// TIA Portal V18 export
FUNCTION_BLOCK "00_Push-Button_Input"   // FB9, F_LAD
{ S7_Optimized_Access := 'TRUE' }
   VAR_INPUT
      Bypass_ET200 : Bool;
      IN_1 : Bool;
      IN_2 : Bool;
      IN_3 : Bool;
      IN_4 : Bool;
      ON_Tristate : Bool;
      NormOpenDiag : Bool;   // if 1-> diag has NO logic, if 0 diag has NC logic
      ON_Lamp : Bool;
      RESET : Bool;
      REAC_DELAY { ExternalWritable := 'False'} : Time;   // Reactivation delay= the OUT goes from 0 to 1 after this time
      BLINK_CYCLE_TIME : Time := t#1250ms;
      ON_TIME : Time := T#625ms;
   END_VAR
   VAR_OUTPUT
      OUT_1 : Bool;
      OUT_2 : Bool;
      OUT_3 : Bool;
      OUT_4 : Bool;
      Diag_1 : Bool;
      Diag_2 : Bool;
      Diag_3 : Bool;
      Diag_4 : Bool;
      Lamp_1 : Bool;
      Lamp_2 : Bool;
      Lamp_3 : Bool;
      Lamp_4 : Bool;
   END_VAR
   VAR
      TON_1 { ExternalWritable := 'False'} : TON;
      TON_2 { ExternalWritable := 'False'} : TON;
      TON_3 { ExternalWritable := 'False'} : TON;
      TON_4 { ExternalWritable := 'False'} : TON;
      TOF_Lamp1 : TOF;
      TOF_Lamp2 : TOF;
      TOF_Lamp3 : TOF;
      TOF_Lamp4 : TOF;
      PRESSED_1 : Bool;
      PRESSED_2 : Bool;
      PRESSED_3 : Bool;
      PRESSED_4 : Bool;
      s_IN_1_P : Bool;
      s_IN_2_P : Bool;
      s_IN_3_P : Bool;
      s_IN_4_P : Bool;
      s_IN_1_N : Bool;
      s_IN_2_N : Bool;
      s_IN_3_N : Bool;
      s_IN_4_N : Bool;
      DUTY_CYCLE : Time;
   END_VAR
   VAR_TEMP
      t_IN1 : Bool;
      t_IN2 : Bool;
      t_IN3 : Bool;
      t_IN4 : Bool;
      t_Lamp1 : Bool;
      t_Lamp2 : Bool;
      t_Lamp3 : Bool;
      t_Lamp4 : Bool;
      t_Diag1 : Bool;
      t_Diag2 : Bool;
      t_Diag3 : Bool;
      t_Diag4 : Bool;
   END_VAR
   VAR_TEMP   // added for the SCL form of the ladder/FBD networks
      _w1 : Bool;
      _w2 : Bool;
   END_VAR
BEGIN

REGION Network 1: OUT 1 & Lamp 1
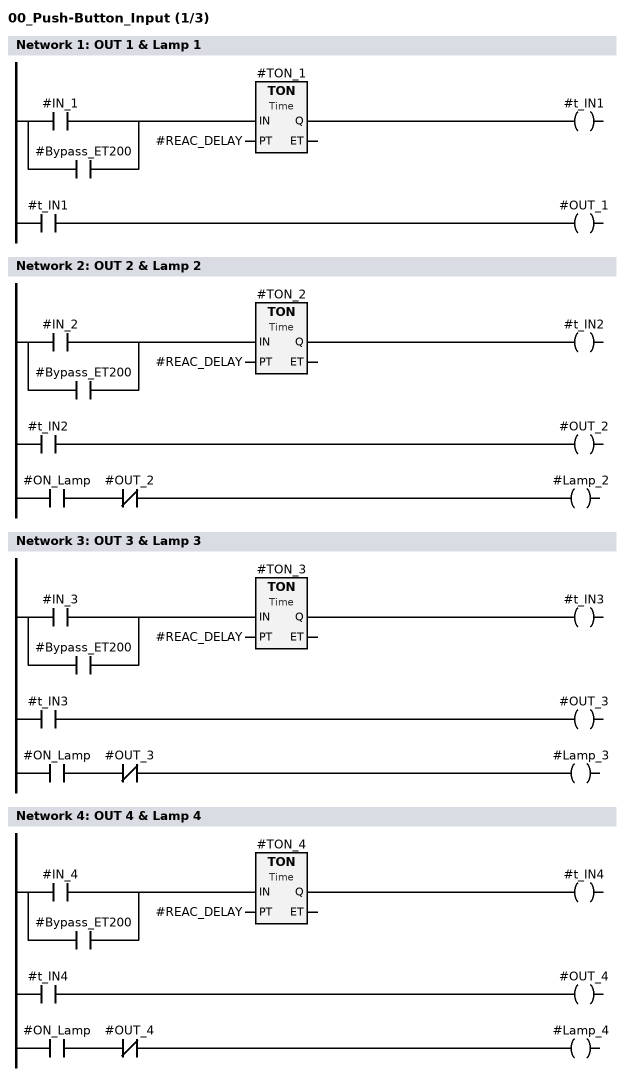
   RUNG wire#powerrail
      Contact( #IN_1 )
      wire#w1
      { S7_Templates := "[time_type := Time, codedbool_type := DInt]" } #TON_1.TON(pt := #REAC_DELAY, et =>)
      Coil( #t_IN1 )
   END_RUNG
   RUNG wire#powerrail
      Contact( #Bypass_ET200 )
   END_RUNG wire#w1
   RUNG wire#powerrail
      Contact( #t_IN1 )
      Coil( #OUT_1 )
   END_RUNG
   // the same network as SCL:
   #TON_1.TON(IN := #IN_1 OR #Bypass_ET200, PT := #REAC_DELAY);
   #t_IN1 := #TON_1.Q;
   #OUT_1 := #t_IN1;
END_REGION

REGION Network 2: OUT 2 & Lamp 2
   RUNG wire#powerrail
      Contact( #IN_2 )
      wire#w1
      { S7_Templates := "[time_type := Time, codedbool_type := DInt]" } #TON_2.TON(pt := #REAC_DELAY, et =>)
      Coil( #t_IN2 )
   END_RUNG
   RUNG wire#powerrail
      Contact( #Bypass_ET200 )
   END_RUNG wire#w1
   RUNG wire#powerrail
      Contact( #t_IN2 )
      Coil( #OUT_2 )
   END_RUNG
   RUNG wire#powerrail
      Contact( #ON_Lamp )
      I_Contact( #OUT_2 )
      Coil( #Lamp_2 )
   END_RUNG
   // the same network as SCL:
   #TON_2.TON(IN := #IN_2 OR #Bypass_ET200, PT := #REAC_DELAY);
   #t_IN2 := #TON_2.Q;
   #OUT_2 := #t_IN2;
   #Lamp_2 := #ON_Lamp AND NOT #OUT_2;
END_REGION

REGION Network 3: OUT 3 & Lamp 3
   RUNG wire#powerrail
      Contact( #IN_3 )
      wire#w1
      { S7_Templates := "[time_type := Time, codedbool_type := DInt]" } #TON_3.TON(pt := #REAC_DELAY, et =>)
      Coil( #t_IN3 )
   END_RUNG
   RUNG wire#powerrail
      Contact( #Bypass_ET200 )
   END_RUNG wire#w1
   RUNG wire#powerrail
      Contact( #t_IN3 )
      Coil( #OUT_3 )
   END_RUNG
   RUNG wire#powerrail
      Contact( #ON_Lamp )
      I_Contact( #OUT_3 )
      Coil( #Lamp_3 )
   END_RUNG
   // the same network as SCL:
   #TON_3.TON(IN := #IN_3 OR #Bypass_ET200, PT := #REAC_DELAY);
   #t_IN3 := #TON_3.Q;
   #OUT_3 := #t_IN3;
   #Lamp_3 := #ON_Lamp AND NOT #OUT_3;
END_REGION

REGION Network 4: OUT 4 & Lamp 4
   RUNG wire#powerrail
      Contact( #IN_4 )
      wire#w1
      { S7_Templates := "[time_type := Time, codedbool_type := DInt]" } #TON_4.TON(pt := #REAC_DELAY, et =>)
      Coil( #t_IN4 )
   END_RUNG
   RUNG wire#powerrail
      Contact( #Bypass_ET200 )
   END_RUNG wire#w1
   RUNG wire#powerrail
      Contact( #t_IN4 )
      Coil( #OUT_4 )
   END_RUNG
   RUNG wire#powerrail
      Contact( #ON_Lamp )
      I_Contact( #OUT_4 )
      Coil( #Lamp_4 )
   END_RUNG
   // the same network as SCL:
   #TON_4.TON(IN := #IN_4 OR #Bypass_ET200, PT := #REAC_DELAY);
   #t_IN4 := #TON_4.Q;
   #OUT_4 := #t_IN4;
   #Lamp_4 := #ON_Lamp AND NOT #OUT_4;
END_REGION

REGION Network 5: Diag 1
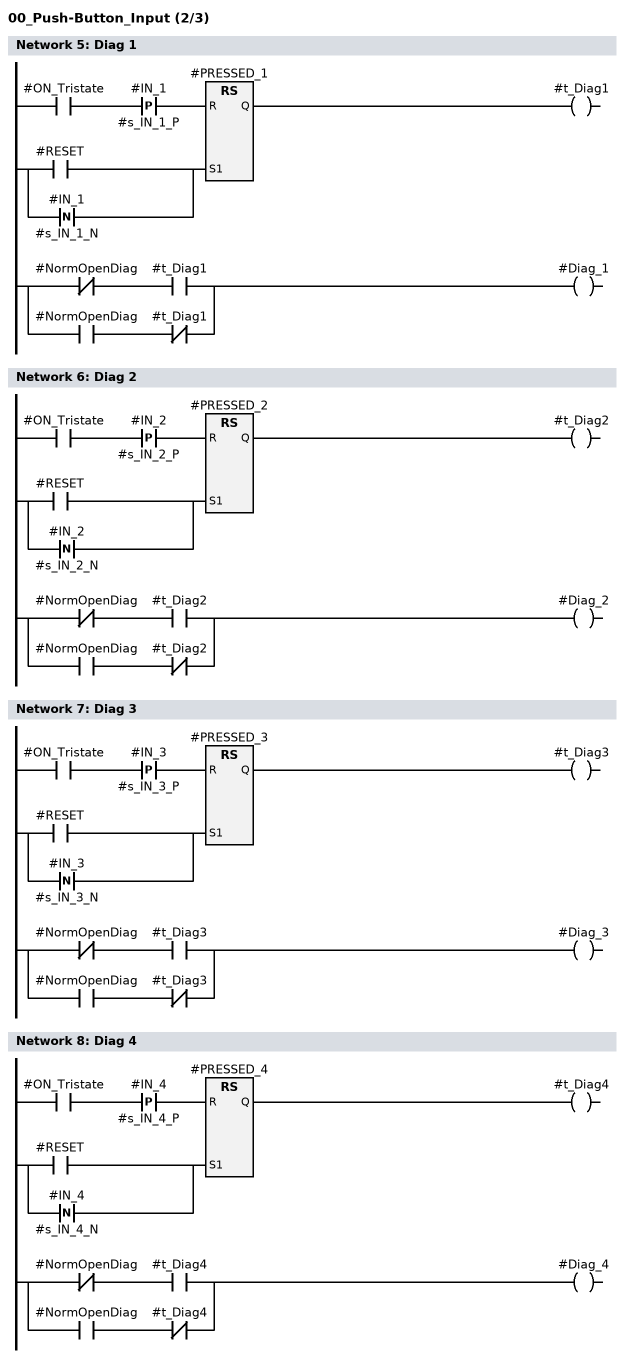
   RUNG wire#powerrail
      Contact( #ON_Tristate )
      P_Contact(operand := #IN_1, bit := #s_IN_1_P)
      S_RS(operand := #PRESSED_1, s1 := wire#w1)
      Coil( #t_Diag1 )
   END_RUNG
   RUNG wire#powerrail
      Contact( #RESET )
   END_RUNG wire#w1
   RUNG wire#powerrail
      N_Contact(operand := #IN_1, bit := #s_IN_1_N)
   END_RUNG wire#w1
   RUNG wire#powerrail
      I_Contact( #NormOpenDiag )
      Contact( #t_Diag1 )
      wire#w2
      Coil( #Diag_1 )
   END_RUNG
   RUNG wire#powerrail
      Contact( #NormOpenDiag )
      I_Contact( #t_Diag1 )
   END_RUNG wire#w2
   // the same network as SCL:
   #_w1 := #ON_Tristate AND #IN_1 AND NOT #s_IN_1_P;   // rising edge of #IN_1
   #s_IN_1_P := #IN_1;
   #_w2 := NOT #IN_1 AND #s_IN_1_N;   // falling edge of #IN_1
   #s_IN_1_N := #IN_1;
   IF #_w1 THEN
       #PRESSED_1 := FALSE;   // RS flip-flop
   END_IF;
   IF #RESET OR #_w2 THEN #PRESSED_1 := TRUE; END_IF;
   #t_Diag1 := #PRESSED_1;
   #Diag_1 := (NOT #NormOpenDiag AND #t_Diag1) OR (#NormOpenDiag AND NOT #t_Diag1);
END_REGION

REGION Network 6: Diag 2
   RUNG wire#powerrail
      Contact( #ON_Tristate )
      P_Contact(operand := #IN_2, bit := #s_IN_2_P)
      S_RS(operand := #PRESSED_2, s1 := wire#w1)
      Coil( #t_Diag2 )
   END_RUNG
   RUNG wire#powerrail
      Contact( #RESET )
   END_RUNG wire#w1
   RUNG wire#powerrail
      N_Contact(operand := #IN_2, bit := #s_IN_2_N)
   END_RUNG wire#w1
   RUNG wire#powerrail
      I_Contact( #NormOpenDiag )
      Contact( #t_Diag2 )
      wire#w2
      Coil( #Diag_2 )
   END_RUNG
   RUNG wire#powerrail
      Contact( #NormOpenDiag )
      I_Contact( #t_Diag2 )
   END_RUNG wire#w2
   // the same network as SCL:
   #_w1 := #ON_Tristate AND #IN_2 AND NOT #s_IN_2_P;   // rising edge of #IN_2
   #s_IN_2_P := #IN_2;
   #_w2 := NOT #IN_2 AND #s_IN_2_N;   // falling edge of #IN_2
   #s_IN_2_N := #IN_2;
   IF #_w1 THEN
       #PRESSED_2 := FALSE;   // RS flip-flop
   END_IF;
   IF #RESET OR #_w2 THEN #PRESSED_2 := TRUE; END_IF;
   #t_Diag2 := #PRESSED_2;
   #Diag_2 := (NOT #NormOpenDiag AND #t_Diag2) OR (#NormOpenDiag AND NOT #t_Diag2);
END_REGION

REGION Network 7: Diag 3
   RUNG wire#powerrail
      Contact( #ON_Tristate )
      P_Contact(operand := #IN_3, bit := #s_IN_3_P)
      S_RS(operand := #PRESSED_3, s1 := wire#w1)
      Coil( #t_Diag3 )
   END_RUNG
   RUNG wire#powerrail
      Contact( #RESET )
   END_RUNG wire#w1
   RUNG wire#powerrail
      N_Contact(operand := #IN_3, bit := #s_IN_3_N)
   END_RUNG wire#w1
   RUNG wire#powerrail
      I_Contact( #NormOpenDiag )
      Contact( #t_Diag3 )
      wire#w2
      Coil( #Diag_3 )
   END_RUNG
   RUNG wire#powerrail
      Contact( #NormOpenDiag )
      I_Contact( #t_Diag3 )
   END_RUNG wire#w2
   // the same network as SCL:
   #_w1 := #ON_Tristate AND #IN_3 AND NOT #s_IN_3_P;   // rising edge of #IN_3
   #s_IN_3_P := #IN_3;
   #_w2 := NOT #IN_3 AND #s_IN_3_N;   // falling edge of #IN_3
   #s_IN_3_N := #IN_3;
   IF #_w1 THEN
       #PRESSED_3 := FALSE;   // RS flip-flop
   END_IF;
   IF #RESET OR #_w2 THEN #PRESSED_3 := TRUE; END_IF;
   #t_Diag3 := #PRESSED_3;
   #Diag_3 := (NOT #NormOpenDiag AND #t_Diag3) OR (#NormOpenDiag AND NOT #t_Diag3);
END_REGION

REGION Network 8: Diag 4
   RUNG wire#powerrail
      Contact( #ON_Tristate )
      P_Contact(operand := #IN_4, bit := #s_IN_4_P)
      S_RS(operand := #PRESSED_4, s1 := wire#w1)
      Coil( #t_Diag4 )
   END_RUNG
   RUNG wire#powerrail
      Contact( #RESET )
   END_RUNG wire#w1
   RUNG wire#powerrail
      N_Contact(operand := #IN_4, bit := #s_IN_4_N)
   END_RUNG wire#w1
   RUNG wire#powerrail
      I_Contact( #NormOpenDiag )
      Contact( #t_Diag4 )
      wire#w2
      Coil( #Diag_4 )
   END_RUNG
   RUNG wire#powerrail
      Contact( #NormOpenDiag )
      I_Contact( #t_Diag4 )
   END_RUNG wire#w2
   // the same network as SCL:
   #_w1 := #ON_Tristate AND #IN_4 AND NOT #s_IN_4_P;   // rising edge of #IN_4
   #s_IN_4_P := #IN_4;
   #_w2 := NOT #IN_4 AND #s_IN_4_N;   // falling edge of #IN_4
   #s_IN_4_N := #IN_4;
   IF #_w1 THEN
       #PRESSED_4 := FALSE;   // RS flip-flop
   END_IF;
   IF #RESET OR #_w2 THEN #PRESSED_4 := TRUE; END_IF;
   #t_Diag4 := #PRESSED_4;
   #Diag_4 := (NOT #NormOpenDiag AND #t_Diag4) OR (#NormOpenDiag AND NOT #t_Diag4);
END_REGION

REGION Network 10: Lamp 1
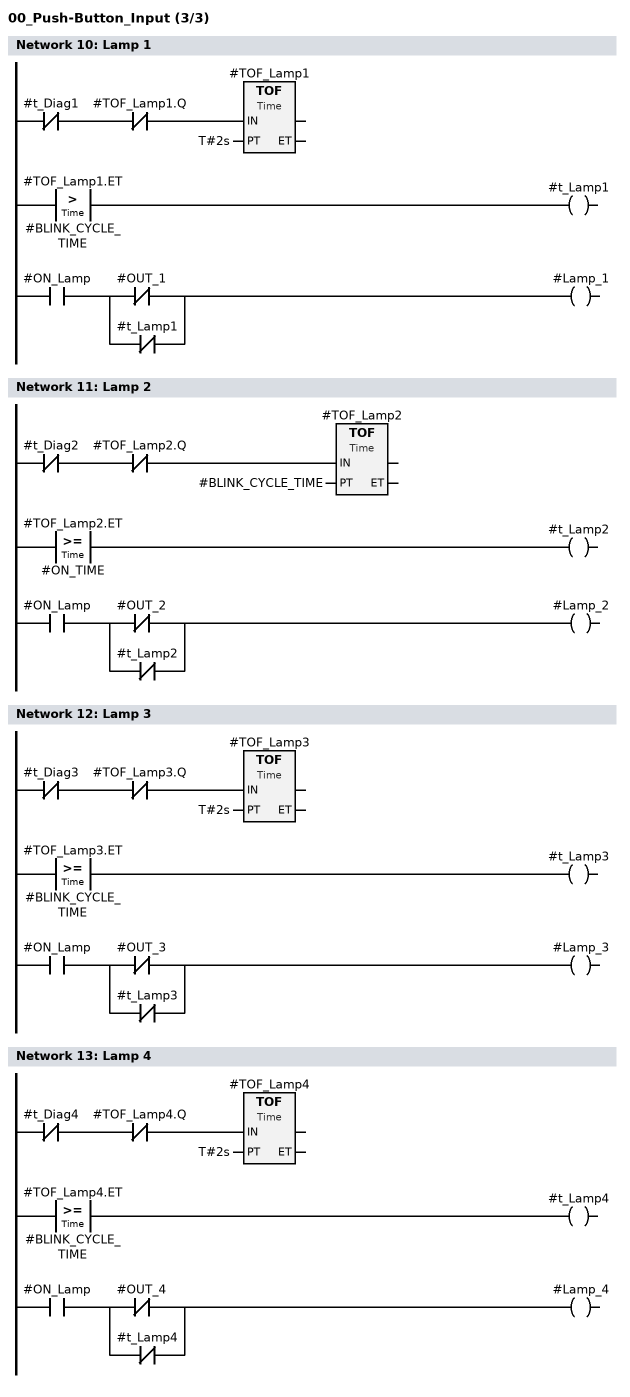
   RUNG wire#powerrail
      I_Contact( #t_Diag1 )
      I_Contact( #TOF_Lamp1.Q )
      { S7_Templates := "[time_type := Time, codedbool_type := DInt]" } #TOF_Lamp1.TOF(pt := T#2s, et =>)
   END_RUNG
   RUNG wire#powerrail
      { S7_Templates := "SrcType := Time" } GT_Contact(in1 := #TOF_Lamp1.ET, in2 := #BLINK_CYCLE_TIME)
      Coil( #t_Lamp1 )
   END_RUNG
   RUNG wire#powerrail
      Contact( #ON_Lamp )
      wire#w1
      I_Contact( #OUT_1 )
      wire#w2
      Coil( #Lamp_1 )
   END_RUNG
   RUNG wire#w1
      I_Contact( #t_Lamp1 )
   END_RUNG wire#w2
   // the same network as SCL:
   #TOF_Lamp1.TOF(IN := NOT #t_Diag1 AND NOT #TOF_Lamp1.Q, PT := T#2s);
   #t_Lamp1 := #TOF_Lamp1.ET > #BLINK_CYCLE_TIME;
   #Lamp_1 := #ON_Lamp AND (NOT #OUT_1 OR NOT #t_Lamp1);
END_REGION

REGION Network 11: Lamp 2
   RUNG wire#powerrail
      I_Contact( #t_Diag2 )
      I_Contact( #TOF_Lamp2.Q )
      { S7_Templates := "[time_type := Time, codedbool_type := DInt]" } #TOF_Lamp2.TOF(pt := #BLINK_CYCLE_TIME, et =>)
   END_RUNG
   RUNG wire#powerrail
      { S7_Templates := "SrcType := Time" } GE_Contact(in1 := #TOF_Lamp2.ET, in2 := #ON_TIME)
      Coil( #t_Lamp2 )
   END_RUNG
   RUNG wire#powerrail
      Contact( #ON_Lamp )
      wire#w1
      I_Contact( #OUT_2 )
      wire#w2
      Coil( #Lamp_2 )
   END_RUNG
   RUNG wire#w1
      I_Contact( #t_Lamp2 )
   END_RUNG wire#w2
   // the same network as SCL:
   #TOF_Lamp2.TOF(IN := NOT #t_Diag2 AND NOT #TOF_Lamp2.Q, PT := #BLINK_CYCLE_TIME);
   #t_Lamp2 := #TOF_Lamp2.ET >= #ON_TIME;
   #Lamp_2 := #ON_Lamp AND (NOT #OUT_2 OR NOT #t_Lamp2);
END_REGION

REGION Network 12: Lamp 3
   RUNG wire#powerrail
      I_Contact( #t_Diag3 )
      I_Contact( #TOF_Lamp3.Q )
      { S7_Templates := "[time_type := Time, codedbool_type := DInt]" } #TOF_Lamp3.TOF(pt := T#2s, et =>)
   END_RUNG
   RUNG wire#powerrail
      { S7_Templates := "SrcType := Time" } GE_Contact(in1 := #TOF_Lamp3.ET, in2 := #BLINK_CYCLE_TIME)
      Coil( #t_Lamp3 )
   END_RUNG
   RUNG wire#powerrail
      Contact( #ON_Lamp )
      wire#w1
      I_Contact( #OUT_3 )
      wire#w2
      Coil( #Lamp_3 )
   END_RUNG
   RUNG wire#w1
      I_Contact( #t_Lamp3 )
   END_RUNG wire#w2
   // the same network as SCL:
   #TOF_Lamp3.TOF(IN := NOT #t_Diag3 AND NOT #TOF_Lamp3.Q, PT := T#2s);
   #t_Lamp3 := #TOF_Lamp3.ET >= #BLINK_CYCLE_TIME;
   #Lamp_3 := #ON_Lamp AND (NOT #OUT_3 OR NOT #t_Lamp3);
END_REGION

REGION Network 13: Lamp 4
   RUNG wire#powerrail
      I_Contact( #t_Diag4 )
      I_Contact( #TOF_Lamp4.Q )
      { S7_Templates := "[time_type := Time, codedbool_type := DInt]" } #TOF_Lamp4.TOF(pt := T#2s, et =>)
   END_RUNG
   RUNG wire#powerrail
      { S7_Templates := "SrcType := Time" } GE_Contact(in1 := #TOF_Lamp4.ET, in2 := #BLINK_CYCLE_TIME)
      Coil( #t_Lamp4 )
   END_RUNG
   RUNG wire#powerrail
      Contact( #ON_Lamp )
      wire#w1
      I_Contact( #OUT_4 )
      wire#w2
      Coil( #Lamp_4 )
   END_RUNG
   RUNG wire#w1
      I_Contact( #t_Lamp4 )
   END_RUNG wire#w2
   // the same network as SCL:
   #TOF_Lamp4.TOF(IN := NOT #t_Diag4 AND NOT #TOF_Lamp4.Q, PT := T#2s);
   #t_Lamp4 := #TOF_Lamp4.ET >= #BLINK_CYCLE_TIME;
   #Lamp_4 := #ON_Lamp AND (NOT #OUT_4 OR NOT #t_Lamp4);
END_REGION
END_FUNCTION_BLOCK
